PROGRAM S11_Packing
VAR
END_VAR

A_Input();
Alarm();
Delay();
FlowAuto();
FlowInit();
General();
ILC();
TipAuto();
TipManual();
Z_Output();

END_PROGRAM

(* stored: Version 1.1.0.1, ProductVersion 3.1.4024.9
   POU S11_Packing: Id {4bfd7582-f391-4d01-b44f-102e87306b7f}, SpecialFunc None *)
